{attribute 'GeneratedUsingTerminal: EL2535-0103-0023'}
{attribute addProperty BoxType "EL2535-0103-0023"}
{attribute addProperty Id "PWM_Status_Channel_1AT %I*PWM_Status_Channel_77939B114PWM_Status_Channel_2AT %I*PWM_Status_Channel_77939B114PWM_Control_Channel_1AT %Q*PWM_Control_Channel_63F162E45PWM_Control_Channel_2AT %Q*PWM_Control_Channel_63F162E45WcStateAT %I*WcState_9091E0EB2InfoDataAT %I*InfoData_94A18F5E2"}
{attribute addProperty CRC "734138001"}
{attribute addProperty Size "22"}
TYPE EL2535_2BC20E91 EXTENDS EtcSlaveTerminalBase_947E5A46 :
STRUCT
	{attribute addProperty Name "PWM_Status_Channel_1"}
	PWM_Status_Channel_1 : PWM_Status_Channel_77939B11;
	{attribute addProperty Name "PWM_Status_Channel_2"}
	PWM_Status_Channel_2 : PWM_Status_Channel_77939B11;
	{attribute addProperty Name "PWM_Control_Channel_1"}
	PWM_Control_Channel_1 : PWM_Control_Channel_63F162E4;
	{attribute addProperty Name "PWM_Control_Channel_2"}
	PWM_Control_Channel_2 : PWM_Control_Channel_63F162E4;
	{attribute addProperty Name "WcState"}
	WcState : WcState_9091E0EB;
	{attribute addProperty Name "InfoData"}
	InfoData : InfoData_94A18F5E;
END_STRUCT
END_TYPE

(* stored: Version 1.2.0.0, ProductVersion 3.1.4024.9
   DUT EL2535_2BC20E91: Id {88b1c07c-40b4-4879-b6ff-bd538b898ade} *)
